(* PLC project Unnamed, Неизвестно Unnamed 1 *)
(* stored: creationDateTime 2024-08-29T09:00:08, modificationDateTime 2024-09-23T10:19:55 *)

TYPE datatype3 : (firstType, secondType) := firstType;
END_TYPE

TYPE datatype0 : ARRAY[10..20, 50..60] OF WORD := [1, 1];
END_TYPE

TYPE datatype1 : INT(0..0) := 0;
END_TYPE

TYPE datatype2 : SINT(0..0) := 0;
END_TYPE

TYPE datatype4 : USINT(0..0) := 0;
END_TYPE

TYPE datatype5 : STRUCT
  p0 : datatype3;
  p1 : DINT;
  p2 : DINT;
  p3 : DINT;
END_STRUCT;
END_TYPE

TYPE datatype6 : TIME;
END_TYPE

PROGRAM program01
  VAR
    IN_0 : BOOL := TRUE;
    IN_OUT_25 : BOOL := TRUE;
    IN_OUT_26 : UINT := 0;
    IN_OUT_27 : REAL := 2.7;
    IN_1 : BOOL := TRUE;
    OUT_0 : BOOL;
    IN_2 : BOOL;
    IN_22 : BOOL := FALSE;
    IN_23 : BOOL := FALSE;
    IN_24 : BOOL := FALSE;
    IN_3 : REAL := 3.1415926535;
    IN_4 : TIME;
    IN_5 : BOOL;
    IN_6 : REAL := 3.1415926535;
    IN_7 : UINT;
    IN_8 : UINT;
    IN_9 : DT;
    IN_10 : TIME;
    IN_11 : BYTE;
    IN_12 : INT;
    IN_13 : DWORD;
    IN_14 : DWORD;
    IN_15 : LREAL;
    IN_16 : LREAL;
    IN_17 : LREAL;
    IN_18 : LREAL;
    IN_19 : LREAL;
    IN_20 : STRING := 'Hello';
    IN_21 : STRING := 'HELLO';
    OUT_1 : REAL;
    OUT_2 : SINT;
    OUT_3 : REAL;
    OUT_4 : UINT;
    OUT_5 : DT;
    OUT_6 : BYTE;
    OUT_7 : DWORD;
    OUT_8 : LREAL;
    OUT_9 : BOOL;
    OUT_10 : STRING;
    LOC_ARR_VAR : datatype5;
    LOC_EN_VAR0 : datatype3;
    SEMA0 : SEMA;
    DERIVATIVE0 : DERIVATIVE;
    SEMA1 : SEMA;
    SR0 : SR;
    RS0 : RS;
  END_VAR
  VAR  (* added by the conversion: wires and edge detectors of the diagram *)
    _ROR52_OUT : BYTE;
    _XOR54_OUT : DWORD;
    _MUL46_OUT : UINT;
  END_VAR

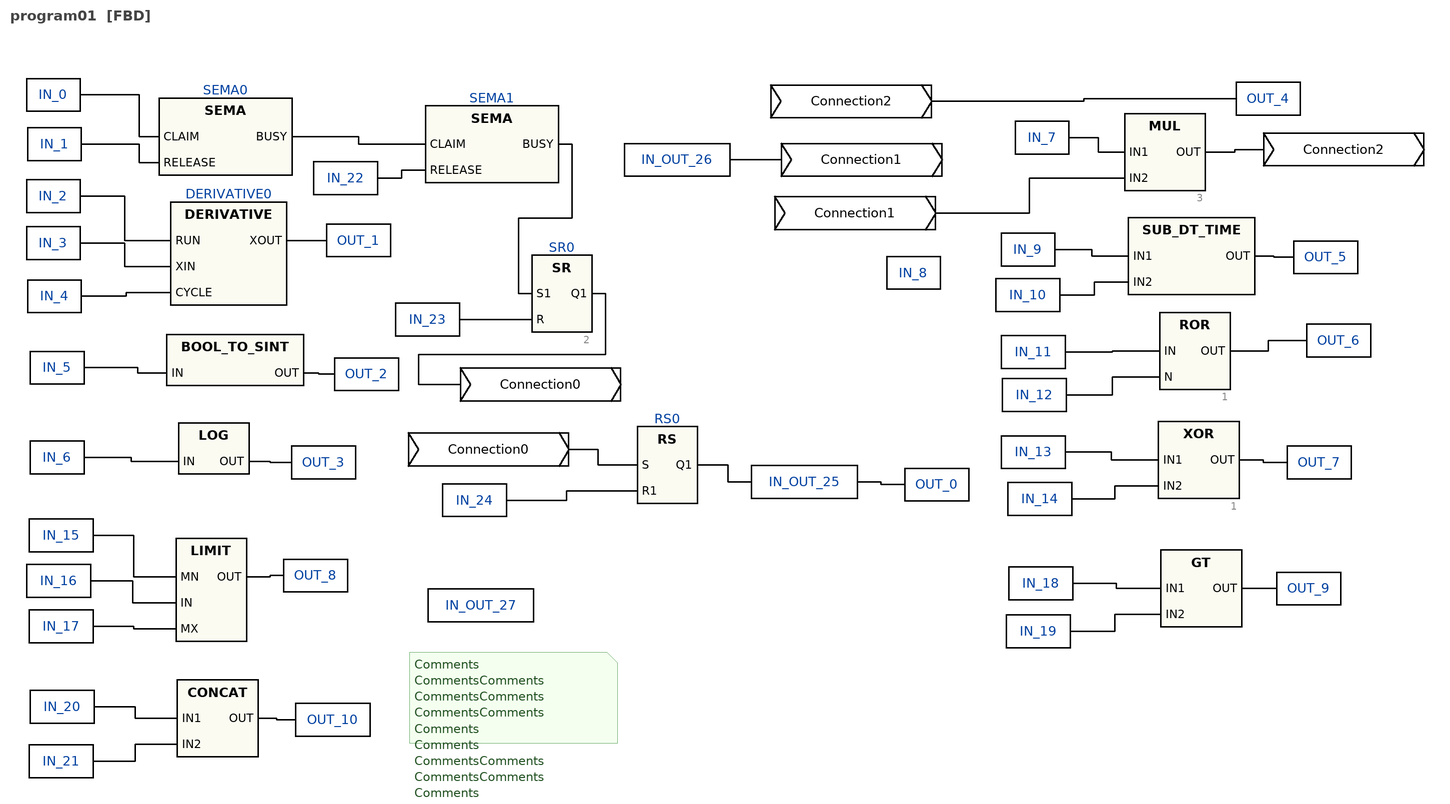
(* FBD diagram, written out as Structured Text *)
_ROR52_OUT := ROR(IN_11, IN_12);
_XOR54_OUT := IN_13 XOR IN_14;
SR0(S1 := SEMA1.BUSY, R := IN_23);
_MUL46_OUT := IN_7 * IN_OUT_26;
DERIVATIVE0(RUN := IN_2, XIN := IN_3, CYCLE := IN_4);
OUT_1 := DERIVATIVE0.XOUT;
OUT_2 := BOOL_TO_SINT(IN_5);
OUT_3 := LOG(IN_6);
OUT_4 := _MUL46_OUT;
OUT_5 := SUB_DT_TIME(IN_9, IN_10);
OUT_6 := _ROR52_OUT;
OUT_7 := _XOR54_OUT;
OUT_8 := LIMIT(IN_15, IN_16, IN_17);
OUT_9 := IN_18 > IN_19;
(* Comments CommentsComments CommentsComments CommentsComments Comments
Comments CommentsComments CommentsComments Comments
Comments CommentsComments CommentsComments Comments
Comments CommentsComments CommentsComments Comments *)
OUT_10 := CONCAT(IN_20, IN_21);
OUT_0 := IN_OUT_25;
RS0(S := SR0.Q1, R1 := IN_24);
IN_OUT_25 := RS0.Q1;
SEMA0(CLAIM := IN_0, RELEASE := IN_1);
SEMA1(CLAIM := SEMA0.BUSY, RELEASE := IN_22);
(* drawn but not wired to any output: IN_8 *)
END_PROGRAM

PROGRAM program0
  VAR
    SEMA0 : SEMA;
    SR0 : SR;
    SR1 : SR;
    RS0 : RS;
    IN_0 : BOOL;
    IN_1 : BOOL;
    IN_2 : BOOL;
    IN_3 : BOOL;
    IN_4 : BOOL;
    OUT_0 : BOOL;
    LOC_ARR_VAR : datatype5;
    LOC_EN_VAR0 : datatype3;
  END_VAR

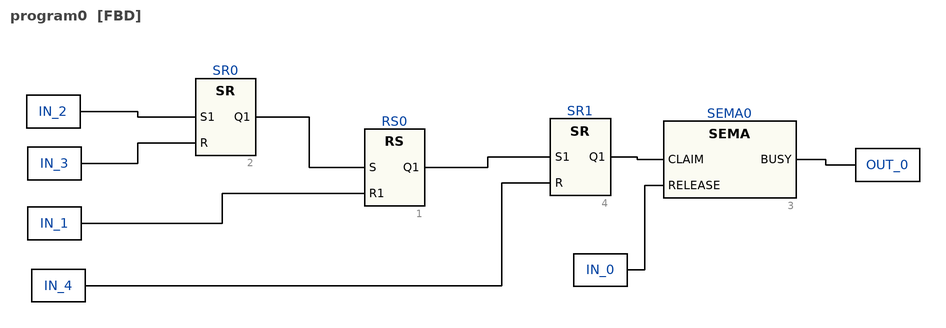
(* FBD diagram, written out as Structured Text *)
RS0(S := SR0.Q1, R1 := IN_1);
SR0(S1 := IN_2, R := IN_3);
SEMA0(CLAIM := SR1.Q1, RELEASE := IN_0);
SR1(S1 := RS0.Q1, R := IN_4);
OUT_0 := SEMA0.BUSY;
END_PROGRAM

CONFIGURATION config
  RESOURCE resource1 ON PLC
    TASK task0(INTERVAL := T#20ms, PRIORITY := 0);
    TASK task1(INTERVAL := T#20ms, PRIORITY := 0);
    PROGRAM instance0 WITH task0 : program0;
    PROGRAM instance1 WITH task1 : program01;
  END_RESOURCE
END_CONFIGURATION
